FUNCTION_BLOCK Test_TLogger_LogError EXTENDS T_UnitTestBase
VAR
    SourceInfo : FB_TcSourceInfo;
END_VAR

{attribute 'analysis' := '-33'} // inhibit unused variable warning
METHOD RunTest
VAR
    ErrorMsg : STRING := 'Expected error message';
END_VAR
IF Retest THEN
    SUPER^.Init();
END_IF

IF TestCompleted THEN
    RETURN;
END_IF

F_Inc(CycleCount);
IF CycleCount > 1000 THEN
    Fail(Message := 'Timeout');
END_IF

SourceInfo.sName := 'ExpectedSourceName';
DefaultLogger.LogError(SourceInfo,'Expected error message1');
DefaultLogger.LogError(SourceInfo,'Expected error message2');

TestCompleted := TRUE;
END_METHOD

END_FUNCTION_BLOCK

(* stored: Version 1.1.0.1, ProductVersion 3.1.4024.15
   POU Test_TLogger_LogError: Id {0d142724-2fcc-4f00-a8dc-b3037bd3c404}, SpecialFunc None
   Method RunTest: Id {51a5d097-350d-4c61-af40-a510294b779f} *)
